{attribute 'qualified_only'}
VAR_GLOBAL
		Device_1_EtherCAT : Device_1_EtherCAT_B557D6C6;
		Device_2_EtherCAT : Device_2_EtherCAT_CA128DDC;
		Device_3_EtherCAT : Device_3_EtherCAT_CA191EDE;
END_VAR

(* stored: Version 1.2.0.0, ProductVersion 3.1.4024.11
   GVL GVL_iXlinker: Id {56e333e8-92a2-4cba-94b7-5db114275511} *)
